FUNCTION_BLOCK ABSTRACT FBA_LinearDrive IMPLEMENTS I_LinearDrive
VAR_INPUT
	bEnable : BOOL;
	sensorDefaultState : BOOL;
END_VAR
VAR_OUTPUT	
	ready : BOOL;
END_VAR
VAR
	direction : MC_Direction;
	
	step : Homing;
	homingComplete : BOOL;
	
	home AT %I* : BOOL;
END_VAR

PROPERTY ABSTRACT Active : BOOL
GET
END_GET
END_PROPERTY

{attribute 'monitoring':='call'}
PROPERTY AtHome : BOOL
GET
AtHome := home <> sensorDefaultState;
END_GET
END_PROPERTY

PROPERTY ABSTRACT Error : BOOL
GET
END_GET
END_PROPERTY

{attribute 'monitoring':='call'}
PROPERTY HomeSet : BOOL
GET
HomeSet := homingComplete;
END_GET
END_PROPERTY

METHOD ABSTRACT homingSequence : BOOL
VAR_INPUT
END_VAR
END_METHOD

METHOD ABSTRACT reset : BOOL
VAR_INPUT
END_VAR
END_METHOD

METHOD ABSTRACT stop : BOOL
VAR_INPUT
END_VAR
END_METHOD

METHOD ABSTRACT toHome : BOOL
VAR_INPUT
END_VAR
END_METHOD

END_FUNCTION_BLOCK

(* stored: Version 1.1.0.1, ProductVersion 3.1.4024.11
   POU FBA_LinearDrive: Id {6e18b76e-a910-410f-9bdc-e9944499ac6c}, SpecialFunc None
   Folder Abstract: Id {5b852458-7492-4207-8a3a-423e79cadb10}
   Folder Properties: Id {020ecba9-69b8-4211-9cef-e7d5a290d286}
   Property Active: Id {13443598-2d95-43e0-9ad5-d28301452e86}
   Get Get: Id {0ab7de27-bc4c-45c1-90b5-180d1941a751}
   Property AtHome: Id {8ff14c6f-db84-4593-a15a-ceabfefdb83b}
   Get Get: Id {b616309b-65d0-4abe-919a-19c39dbec209}
   Property Error: Id {6abbeb83-adc3-4eaf-aa72-9f30d95d101f}
   Get Get: Id {72228712-55ba-4ec3-aad4-a86a30100290}
   Property HomeSet: Id {a698b452-7d02-48c3-95ad-c49887df96f3}
   Get Get: Id {19f25ff9-f621-402b-9154-b013de85f2a1}
   Method homingSequence: Id {960b0ee1-804c-4505-b278-f1901847cba6}
   Method reset: Id {fa731df6-6b1e-4d97-8750-1bb688b2ee7a}
   Method stop: Id {ef1daccc-48c1-47ec-a753-b7db2650175f}
   Method toHome: Id {a50dcacf-df9c-4f3e-8e4d-8625f542db41} *)
